Yaskawa INFORM job: INITIALISATION-I-O.JBI

/JOB
//NAME INITIALISATION-I-O
//POS
///NPOS 0,0,0,0,0,0
//INST
///DATE 2018/08/30 13:15
///ATTR SC,RW
NOP
DOUT OG#(64) 0
DOUT OG#(65) 0
DOUT OG#(66) 0
DOUT OG#(67) 0
DOUT OG#(68) 0
DOUT OG#(69) 0
DOUT OG#(70) 0
DOUT OG#(71) 0
DOUT OG#(72) 0
DOUT OG#(73) 0
DOUT OG#(74) 0
DOUT OG#(75) 0
DOUT OG#(76) 0
DOUT OG#(77) 0
END
